{attribute 'qualified_only'}
{attribute 'strict'}
{attribute 'to_string'}
TYPE mainStateMachineStatus_t :
(
	IDLE := 0,
	ROTATE_TABLE,
	GRIPPER_DOWN,
	GRIPPER_CLOSE,
	GRIPPER_UP,
	GRIPPER_LEFT,
	GRIPPER_DOWN_LEFT,
	GRIPPER_OPEN,
	GRIPPER_UP_LEFT,
	GRIPPER_RIGHT,
	Y10_OUT,
	CONVAYORBELT_START,
	Y10_BACK,
	Y2_OUT,
	Y3_OUT,
	CONVEYORBELT_STOP,
);
END_TYPE

(* stored: Version 1.1.0.1
   EnumerationTextList mainStateMachineStatus_t: Id {dad8ecc4-42e9-4a2a-8d28-578b206aa962} *)
